RoboDK station: Block1.rdk

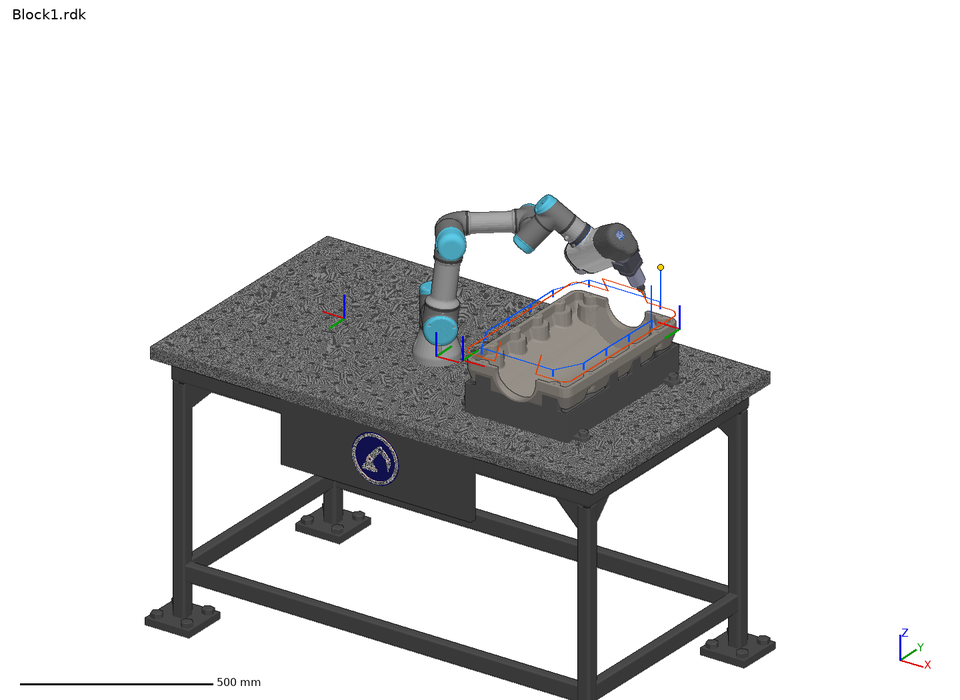
[picture v0: the station drawn from its stored meshes, robots at their saved joint values, targets as dots, program paths as lines]
Station Block1 (saved by RoboDK 5.5.1). Poses are relative to the parent item; angles as X-Y-Z fixed-axis rotations.
Station parameters (name, value as stored): ViewNames, New View 1|[19.806,-223.251,-1852.955,-4.394,-26.413,-81.026]||New View 2|[-145.353,-147.123,-1133.187,-12.666,-29.479,-64.252]||New View 3|[-89.962,-117.618,-1053.622,-35.524,-65.339,-53.555]||New View 4|[104.763,80.763,-3406.264,-32.675,-38.414,-42.423]||, TAGS, ['Dispensing'], Palletizing Plugin
  - frame World at (0, 0, 0) mm
    - object Table at (0, 0, 0) mm, size 1420 x 820 x 800 mm, geometry from Table-1400x800x800.sld
    - frame Doosan Robotics M1013 - Navy Base at (-392.37, 24.39, 0) mm, rotated rx 0 ry 0 rz -180 deg
      - frame Part at (-900, -230, 130) mm
        - object Pan_Holder at (0, 0, 0) mm, size 400 x 503 x 157.6 mm, geometry from Jig2.step
        - object Part_Oil_Pan at (0, 0, 0) mm, size 330.2 x 509.8 x 126.9 mm, 12 curves
  - frame UR3 Base at (-70, -20, 0) mm
    - robot UR3: 6 axes, payload 3 kg, reach 500 mm, repeatability 0.1 mm, weight 11 kg
        modified DH rows (alpha deg, a mm, theta deg, d mm): 0, 0, 0, 151.9; 90, 0, 180, 0; 0, 243.65, 0, 0; 0, 213, 0, 110.4; -90, 0, 0, 83.4; 90, 0, 180, 82.4
        joint limits [-360, -360, -360, -360, -360, -360] to [360, 360, 360, 360, 360, 360]; home [0, -90, -90, 0, 90, 0]; saved at [38.681, -96.552, -82.896, -43.066, 84.837, 137.25]
      - tool Spintech Spindle, TCP at (52, 0, 260) mm, rotated rx 0 ry 39 rz 0 deg, size 157.3 x 72 x 259.9 mm
      - tool OnRobot Screwdriver, TCP at (168.4, 0, 95.37) mm, rotated rx 0 ry 90 rz 0 deg, size 323.9 x 86.2 x 125.3 mm
  - machining project Ajustes de puntos: rotZ(0) | rotX(0)*rotY(0) | rotz(0) | onStart | onPathStart | onApproach | onPoint | onRetract | onFinish | SetRPM(%1) | SetTool(%1) | Extruder(%1) | default | default | OutOnMov(%1) | OutOffMov(%1) | onPathFinish | M_RunCode(%1)
  - program Replace (1 instructions, listed below)
  - program Puntos (71 instructions, listed below)
  - machining project Path2 ajustes curva: rotZ(0) | rotX(0)*rotY(0) | rotz(0) | onStart | onPathStart | onApproach | onPoint | onRetract | onFinish | SetRPM(%1) | SetTool(%1) | Extruder(%1) | default | default | OutOnMov(%1) | OutOffMov(%1) | onPathFinish | M_RunCode(%1)
  - program Main_Program (8 instructions, listed below)
  - program Curva (47 instructions, listed below)
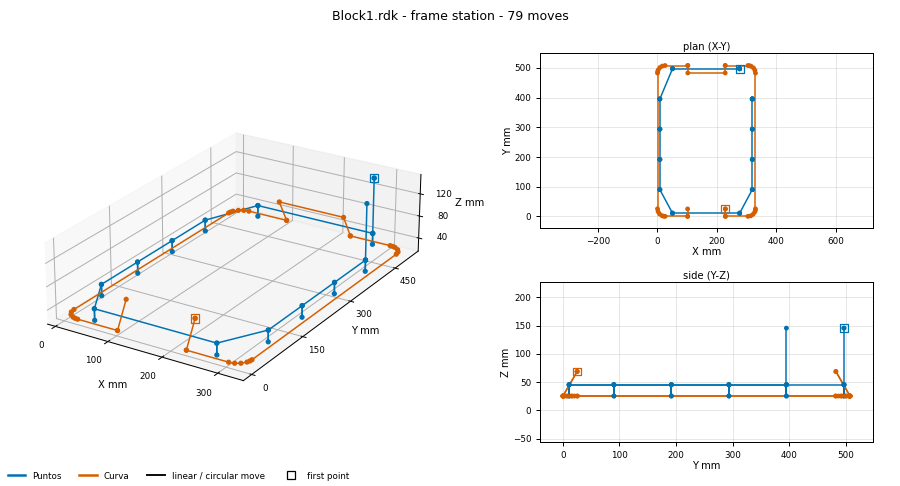
[picture p0: tool path of Block1.rdk in frame station, 79 of 79 moves have a stored position in this frame; points joined in program order, loops and branches not executed]

--- program Replace (robot UR3) ---
  Reemplazar objetos

--- program Puntos (robot UR3) ---
  Suave(1)
  Establecer velocidad (1000.0 mm/s)
  Est. Ref.: World
  Est. herr: OnRobot Screwdriver
  Mostrar OnRobot Screwdriver
  MoveJ 1 to (276.5, 496.76, 145.4) mm, rotated rx -180 ry 0 rz 0 deg; joints [-35.249, -94.444, -94.854, 9.299, 125.249, 90]
  MoveL 2 to (276.5, 496.76, 145.4) mm, rotated rx -180 ry 0 rz 0 deg; joints [-35.249, -94.444, -94.854, 9.299, 125.249, 90]
  MoveL 3 to (276.5, 496.76, 45.4) mm, rotated rx 180 ry 0 rz 0 deg; joints [-35.249, -103.964, -112.957, 36.92, 125.249, 90]
  MoveL 4 to (276.5, 496.76, 45.4) mm, rotated rx 180 ry 0 rz 0 deg; joints [-35.249, -103.964, -112.957, 36.92, 125.249, 90]
  Establecer velocidad (30.0 mm/s)
  MoveL 5 to (276.5, 496.76, 25.4) mm, rotated rx -180 ry 0 rz 0 deg; joints [-35.249, -107.261, -115.34, 42.601, 125.249, 90]
  MoveL 6 to (276.5, 496.76, 45.4) mm, rotated rx 180 ry 0 rz 0 deg; joints [-35.249, -103.964, -112.957, 36.92, 125.249, 90]
  Establecer velocidad (1000.0 mm/s)
  MoveL 7 to (50.77, 496.76, 45.4) mm, rotated rx -180 ry 0 rz 0 deg; joints [-17.027, -141.393, -50.4, 11.793, 107.027, 90]
  Establecer velocidad (30.0 mm/s)
  MoveL 8 to (50.77, 496.76, 25.4) mm, rotated rx -180 ry 0 rz 0 deg; joints [-17.027, -142.831, -53.168, 15.999, 107.027, 90]
  MoveL 9 to (50.77, 496.76, 45.4) mm, rotated rx -180 ry 0 rz 0 deg; joints [-17.027, -141.393, -50.4, 11.793, 107.027, 90]
  Establecer velocidad (1000.0 mm/s)
  MoveL 10 to (8.24, 395.16, 45.4) mm, rotated rx -180 ry 0 rz 0 deg; joints [-1.511, -140.151, -52.768, 12.919, 91.511, 90]
  Establecer velocidad (30.0 mm/s)
  MoveL 11 to (8.24, 395.16, 25.4) mm, rotated rx -180 ry 0 rz 0 deg; joints [-1.511, -141.655, -55.452, 17.108, 91.511, 90]
  MoveL 12 to (8.24, 395.16, 45.4) mm, rotated rx -180 ry 0 rz 0 deg; joints [-1.511, -140.151, -52.768, 12.919, 91.511, 90]
  Establecer velocidad (1000.0 mm/s)
  MoveL 13 to (8.24, 293.56, 45.4) mm, rotated rx -180 ry 0 rz 0 deg; joints [13.552, -135.181, -62.091, 17.272, 76.448, 90]
  Establecer velocidad (30.0 mm/s)
  MoveL 14 to (8.24, 293.56, 25.4) mm, rotated rx -180 ry 0 rz 0 deg; joints [13.552, -136.926, -64.525, 21.452, 76.448, 90]
  MoveL 15 to (8.24, 293.56, 45.4) mm, rotated rx -180 ry 0 rz 0 deg; joints [13.552, -135.181, -62.091, 17.272, 76.448, 90]
  Establecer velocidad (1000.0 mm/s)
  MoveL 16 to (8.24, 191.96, 45.4) mm, rotated rx -180 ry 0 rz 0 deg; joints [27.9, -137.381, -57.995, 15.376, 62.1, 90]
  Establecer velocidad (30.0 mm/s)
  MoveL 17 to (8.24, 191.96, 25.4) mm, rotated rx -180 ry 0 rz 0 deg; joints [27.9, -139.023, -60.526, 19.549, 62.1, 90]
  MoveL 18 to (8.24, 191.96, 45.4) mm, rotated rx -180 ry 0 rz 0 deg; joints [27.9, -137.381, -57.995, 15.376, 62.1, 90]
  Establecer velocidad (1000.0 mm/s)
  MoveL 19 to (8.24, 90.36, 45.4) mm, rotated rx -180 ry 0 rz 0 deg; joints [39.952, -147.907, -37.738, 5.645, 50.048, 90]
  Establecer velocidad (30.0 mm/s)
  MoveL 20 to (8.24, 90.36, 25.4) mm, rotated rx -180 ry 0 rz 0 deg; joints [39.952, -148.919, -41.161, 10.081, 50.048, 90]
  MoveL 21 to (8.24, 90.36, 45.4) mm, rotated rx -180 ry 0 rz 0 deg; joints [39.952, -147.907, -37.738, 5.645, 50.048, 90]
  Establecer velocidad (1000.0 mm/s)
  MoveL 22 to (50.77, 11.24, 45.4) mm, rotated rx -180 ry 0 rz 0 deg; joints [51.637, -149.747, -34.091, 3.838, 38.363, 90]
  Establecer velocidad (30.0 mm/s)
  MoveL 23 to (50.77, 11.24, 25.4) mm, rotated rx -180 ry 0 rz 0 deg; joints [51.637, -150.601, -37.797, 8.397, 38.363, 90]
  MoveL 24 to (50.77, 11.24, 45.4) mm, rotated rx -180 ry 0 rz 0 deg; joints [51.637, -149.747, -34.091, 3.838, 38.363, 90]
  Establecer velocidad (1000.0 mm/s)
  MoveL 25 to (276.5, 11.24, 45.4) mm, rotated rx -180 ry 0 rz 0 deg; joints [87.208, -111.969, -101.496, 33.466, 2.792, 90]
  Establecer velocidad (30.0 mm/s)
  MoveL 26 to (276.5, 11.24, 25.4) mm, rotated rx 180 ry 0 rz 0 deg; joints [87.208, -114.802, -103.725, 38.528, 2.792, 90]
  MoveL 27 to (276.5, 11.24, 45.4) mm, rotated rx -180 ry 0 rz 0 deg; joints [87.208, -111.969, -101.496, 33.466, 2.792, 90]
  Establecer velocidad (1000.0 mm/s)
  MoveL 28 to (319.03, 90.36, 45.4) mm, rotated rx -180 ry 0 rz 20 deg; joints [99.372, -74.581, -141.813, 36.394, 10.628, 90]
  Establecer velocidad (30.0 mm/s)
  MoveL 29 to (319.03, 90.36, 25.4) mm, rotated rx -180 ry 0 rz 20 deg; joints [99.372, -79.77, -145.483, 45.253, 10.628, 90]
  MoveL 30 to (319.03, 90.36, 45.4) mm, rotated rx -180 ry 0 rz 20 deg; joints [99.372, -74.581, -141.813, 36.394, 10.628, 90]
  Establecer velocidad (1000.0 mm/s)
  MoveL 31 to (319.03, 191.96, 45.4) mm, rotated rx -180 ry 0 rz 40 deg; joints [46.203, -58.74, -149.193, 27.933, 83.797, 90]
  Establecer velocidad (30.0 mm/s)
  MoveL 32 to (319.03, 191.96, 25.4) mm, rotated rx -180 ry 0 rz 40 deg; joints [46.203, -64.089, -153.748, 37.836, 83.797, 90]
  MoveL 33 to (319.03, 191.96, 45.4) mm, rotated rx -180 ry 0 rz 40 deg; joints [46.203, -58.74, -149.193, 27.933, 83.797, 90]
  Establecer velocidad (1000.0 mm/s)
  MoveL 34 to (319.03, 293.56, 45.4) mm, rotated rx -180 ry 0 rz 20 deg; joints [24.118, -54.178, -150.538, 24.716, 85.882, 90]
  Establecer velocidad (30.0 mm/s)
  MoveL 35 to (319.03, 293.56, 25.4) mm, rotated rx -180 ry 0 rz 20 deg; joints [24.118, -59.294, -155.319, 34.613, 85.882, 90]
  MoveL 36 to (319.03, 293.56, 45.4) mm, rotated rx -180 ry 0 rz 20 deg; joints [24.118, -54.178, -150.538, 24.716, 85.882, 90]
  Establecer velocidad (1000.0 mm/s)
  MoveL 37 to (319.03, 395.16, 45.4) mm, rotated rx -180 ry 0 rz 0 deg; joints [-6.769, -70.719, -144.056, 34.774, 96.769, 90]
  Establecer velocidad (30.0 mm/s)
  MoveL 38 to (319.03, 395.16, 25.4) mm, rotated rx -180 ry 0 rz 0 deg; joints [-6.769, -76.058, -147.946, 44.004, 96.769, 90]
  MoveL 39 to (319.03, 395.16, 45.4) mm, rotated rx -180 ry 0 rz 0 deg; joints [-6.769, -70.719, -144.056, 34.774, 96.769, 90]
  MoveL 40 to (319.03, 395.16, 45.4) mm, rotated rx -180 ry 0 rz 0 deg; joints [-6.769, -70.719, -144.056, 34.774, 96.769, 90]
  Establecer velocidad (1000.0 mm/s)
  MoveL 41 to (319.03, 395.16, 45.4) mm, rotated rx -180 ry 0 rz 0 deg; joints [-6.769, -70.719, -144.056, 34.774, 96.769, 90]
  MoveL 42 to (319.03, 395.16, 145.4) mm, rotated rx -180 ry 0 rz 0 deg; joints [-6.769, -60.912, -120.277, 1.189, 96.769, 90]

--- program Main_Program (robot UR3) ---
  Llamar Replace
  Ocultar OnRobot Screwdriver
  Mostrar Spintech Spindle
  Llamar Curva
  Pausa 3.0 s
  Ocultar Spintech Spindle
  Mostrar OnRobot Screwdriver
  Llamar Puntos

--- program Curva (robot UR3) ---
  Suave(1)
  Establecer velocidad (1000.0 mm/s)
  Est. Ref.: World
  Est. herr: Spintech Spindle
  Mostrar Spintech Spindle
  MoveJ 1 to (228.6, 25.44, 68.7) mm, rotated rx 150 ry 0 rz 0 deg; joints [63.2, -64.561, -107.739, -54.564, 67.262, 154.952]
  MoveL 2 to (228.6, 25.44, 68.7) mm, rotated rx 150 ry 0 rz 0 deg; joints [63.2, -64.561, -107.739, -54.564, 67.262, 154.952]
  MoveL 3 to (228.6, 0.44, 25.4) mm, rotated rx 150 ry 0 rz 0 deg; joints [66.663, -68.118, -117.167, -42.711, 64.919, 157.742]
  MoveL 4 to (228.6, 0.44, 25.4) mm, rotated rx 150 ry 0 rz 0 deg; joints [66.663, -68.118, -117.167, -42.711, 64.919, 157.742]
  Establecer velocidad (10.0 mm/s)
  MoveL 5 to (304.36, 0.44, 25.4) mm, rotated rx 150.34 ry -4.72 rz 2.69 deg; joints [82.393, -53.535, -117.096, -65.829, 60.419, 172.391]
  MoveL 6 to (313.81, 2.26, 25.4) mm, rotated rx 153.17 ry -13.96 rz 6.96 deg; joints [66.379, -67.029, -103.443, -66.928, 78.266, 158.414]
  MoveL 7 to (321.71, 7.29, 25.4) mm, rotated rx 159.78 ry -22.65 rz 8.07 deg; joints [60.192, -81.14, -83.664, -81.794, 85.879, 151.813]
  MoveL 8 to (327.49, 15.35, 25.4) mm, rotated rx 168.48 ry -27.89 rz 5.45 deg; joints [60.621, -92.638, -65.134, -98.204, 85.669, 151.036]
  MoveL 9 to (329.22, 20.64, 25.4) mm, rotated rx 176.08 ry -29.77 rz 1.95 deg; joints [62.614, -101.614, -50.379, -110.76, 83.416, 152.469]
  MoveL 10 to (329.76, 25.84, 25.4) mm, rotated rx -180 ry -30 rz 0 deg; joints [63.749, -105.614, -43.502, -116.877, 81.935, 153.466]
  MoveL 11 to (329.76, 482.16, 25.4) mm, rotated rx -172.85 ry -29.21 rz -3.5 deg; joints [-13.194, -89.724, -65.735, -103.753, 86.2, 75.923]
  MoveL 12 to (327.94, 491.61, 25.4) mm, rotated rx -161.13 ry -23.76 rz -7.84 deg; joints [-1.252, -75.66, -83.684, -95.62, 73.635, 84.437]
  MoveL 13 to (322.91, 499.51, 25.4) mm, rotated rx -153.87 ry -15.3 rz -7.37 deg; joints [9.756, -59.961, -101.084, -89.075, 63.154, 89.991]
  MoveL 14 to (314.85, 505.29, 25.4) mm, rotated rx -150.95 ry -7.83 rz -4.33 deg; joints [15.987, -47.144, -113.326, -83.721, 57.435, 90.454]
  MoveL 15 to (309.56, 507.02, 25.4) mm, rotated rx -150.1 ry -2.56 rz -1.47 deg; joints [18.883, -37.764, -120.89, -80.031, 55.15, 88.907]
  MoveL 16 to (304.36, 507.56, 25.4) mm, rotated rx -150 ry 0 rz 0 deg; joints [18.335, -34.667, -124.545, -75.567, 55.472, 86.226]
  MoveL 17 to (227.98, 507.56, 25.4) mm, rotated rx -150 ry 0 rz 0 deg; joints [9.13, -61.034, -120.099, -49.12, 61.086, 77.64]
  Establecer velocidad (1000.0 mm/s)
  MoveL 18 to (227.98, 507.56, 25.4) mm, rotated rx -150 ry 0 rz 0 deg; joints [9.13, -61.034, -120.099, -49.12, 61.086, 77.64]
  MoveL 19 to (227.98, 482.56, 68.7) mm, rotated rx -150 ry 0 rz 0 deg; joints [18.22, -58.394, -108.057, -68.263, 55.538, 86.112]
  Establecer velocidad (1000.0 mm/s)
  MoveL 20 to (102.22, 482.56, 68.7) mm, rotated rx -150 ry 0 rz 0 deg; joints [10.076, -91.912, -85.611, -53.138, 60.483, 78.476]
  MoveL 21 to (102.22, 507.56, 25.4) mm, rotated rx -150 ry 0 rz 0 deg; joints [5.154, -94.471, -95.178, -39.023, 63.671, 74.23]
  MoveL 22 to (102.22, 507.56, 25.4) mm, rotated rx -150 ry 0 rz 0 deg; joints [5.154, -94.471, -95.178, -39.023, 63.671, 74.23]
  Establecer velocidad (10.0 mm/s)
  MoveL 23 to (25.84, 507.56, 25.4) mm, rotated rx -150 ry 0 rz 0 deg; joints [4.088, -113.016, -71.689, -43.578, 64.377, 73.342]
  MoveL 24 to (16.39, 505.74, 25.4) mm, rotated rx -150.34 ry 4.72 rz 2.69 deg; joints [2.828, -111.281, -79.767, -31.287, 67.277, 70.388]
  MoveL 25 to (8.49, 500.71, 25.4) mm, rotated rx -153.17 ry 13.96 rz 6.96 deg; joints [-1.854, -109.654, -92.365, -10.341, 76.855, 67.325]
  MoveL 26 to (2.71, 492.65, 25.4) mm, rotated rx -159.78 ry 22.65 rz 8.07 deg; joints [-8.205, -112.15, -97.715, 4.35, 89.065, 69.752]
  MoveL 27 to (0.98, 487.36, 25.4) mm, rotated rx -168.48 ry 27.89 rz 5.45 deg; joints [-13.56, -115.533, -97.626, 10.64, 98.651, 75.435]
  MoveL 28 to (0.44, 482.16, 25.4) mm, rotated rx -176.08 ry 29.77 rz 1.95 deg; joints [-16.579, -117.661, -95.931, 11.755, 104.214, 80.736]
  MoveL 29 to (0.44, 25.84, 25.4) mm, rotated rx -180 ry 30 rz 0 deg; joints [59.273, -119.254, -90.128, -7.535, 36.629, 121.086]
  MoveL 30 to (2.26, 16.39, 25.4) mm, rotated rx 172.85 ry 29.21 rz -3.5 deg; joints [58.475, -118.271, -91.562, -5.285, 39.497, 125.194]
  MoveL 31 to (7.29, 8.49, 25.4) mm, rotated rx 161.13 ry 23.76 rz -7.84 deg; joints [54.238, -114.439, -93.417, -5.776, 49.225, 132.51]
  MoveL 32 to (15.35, 2.71, 25.4) mm, rotated rx 153.87 ry 15.3 rz -7.37 deg; joints [47.444, -111.596, -90.208, -12.775, 63.294, 136.734]
  MoveL 33 to (20.64, 0.98, 25.4) mm, rotated rx 150.95 ry 7.83 rz -4.33 deg; joints [40.661, -112.566, -81.832, -22.824, 76.159, 136.771]
  MoveL 34 to (25.84, 0.44, 25.4) mm, rotated rx 150.1 ry 2.56 rz -1.47 deg; joints [36.448, -115.013, -73.038, -32.352, 84.307, 135.492]
  MoveL 35 to (101.6, 0.44, 25.4) mm, rotated rx 150 ry 0 rz 0 deg; joints [42.292, -99.547, -91.055, -32.19, 82.182, 139.712]
  Establecer velocidad (1000.0 mm/s)
  MoveL 36 to (101.6, 0.44, 25.4) mm, rotated rx 150 ry 0 rz 0 deg; joints [42.292, -99.547, -91.055, -32.19, 82.182, 139.712]
  MoveL 37 to (101.6, 25.44, 68.7) mm, rotated rx 150 ry 0 rz 0 deg; joints [38.681, -96.552, -82.896, -43.066, 84.837, 137.25]
